Staubli VAL3: onF1Event.pgx

program onF1Event(string x_sProg (dimensions=1))
  local string l_sPath
  local num l_nPath
begin
  // look if the bButton is enable
  if bButton[0]
    //
    // go to the edit program
    //
    l_sPath=prog:libPath()+"/page_viewInstr"
    call loadPage(l_sPath,x_sProg)
  endIf
end
